TYPE ST_ServiceCtrl :
STRUCT
	RequestId : UDINT;
	PackMLIn : ST_PML_Base_In;
END_STRUCT
END_TYPE

(* stored: Version 1.1.0.1, ProductVersion 3.1.4026.18
   DUT ST_ServiceCtrl: Id {e3e054b0-1445-4490-9ce3-3d180aa7d013} *)
